FUNCTION Between : BOOL
VAR_INPUT
	in			: REAL;
	lim1		: REAL;
	lim2		: REAL;
END_VAR
VAR
END_VAR

IF lim1 > lim2 THEN 
		IF (in <= lim1) AND (in >= lim2) THEN
			Between:=TRUE;
		ELSE
			Between:=FALSE;
		END_IF

ELSE
		IF (in >= lim1) AND (in <= lim2) THEN
			Between:=TRUE;
		ELSE
			Between:=FALSE;
		END_IF	
END_IF

END_FUNCTION

(* stored: Version 1.1.0.1, ProductVersion 3.1.4026.18
   POU Between: Id {9ea815f3-b71d-45b2-a57e-f4c636ed6f62}, SpecialFunc None *)
